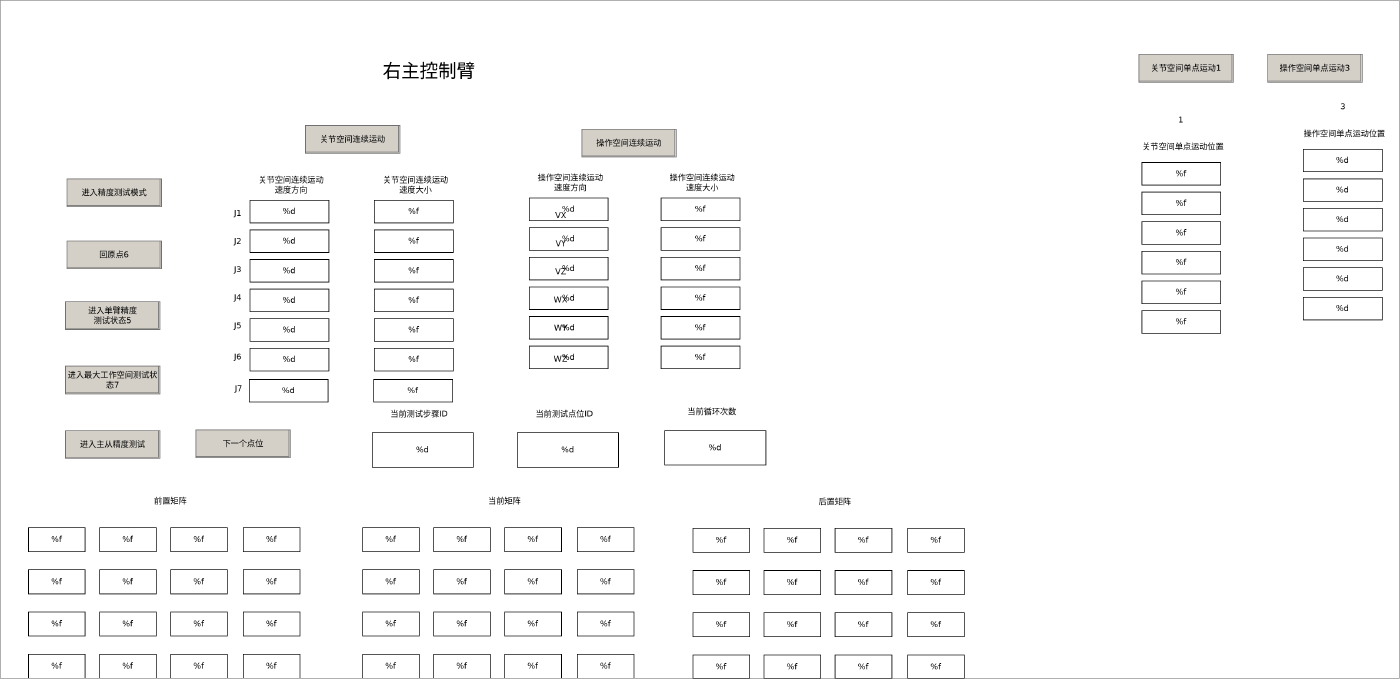
VISUALIZATION Robot_Jog_Arm2_1  // 1890x917
    Label (504,74 150x43), "右主控制臂"
    Rectangle (337,270 107x31), "%d", text variable: GVL_AccuracyTestVar.g_jntMotionDir[2][1]
        OnMouseClick: write the text variable via Default, min -1, max 1
    Label (318,235 150x29), "关节空间连续运动 速度方向"
    Rectangle (337,310 107x31), "%d", text variable: GVL_AccuracyTestVar.g_jntMotionDir[2][2]
        OnMouseClick: write the text variable via Default, min -1, max 1
    Rectangle (337,350 107x31), "%d", text variable: GVL_AccuracyTestVar.g_jntMotionDir[2][3]
        OnMouseClick: write the text variable via Default, min -1, max 1
    Rectangle (337,390 107x31), "%d", text variable: GVL_AccuracyTestVar.g_jntMotionDir[2][4]
        OnMouseClick: write the text variable via Default, min -1, max 1
    Rectangle (337,430 107x31), "%d", text variable: GVL_AccuracyTestVar.g_jntMotionDir[2][5]
        OnMouseClick: write the text variable via Default, min -1, max 1
    Rectangle (337,470 107x31), "%d", text variable: GVL_AccuracyTestVar.g_jntMotionDir[2][6]
        OnMouseClick: write the text variable via Default, min -1, max 1
    Group (1519,147 153x303), invisible if: TRUE
        Rectangle (22,72 107x31), "%f", text variable: GVL_AccuracyTestVar.g_targetJntPos[2][1]
            OnMouseClick: write the text variable via Default
        Label (3,36 150x30), "关节空间单点运动位置"
        Rectangle (22,112 107x31), "%f", text variable: GVL_AccuracyTestVar.g_targetJntPos[2][2]
            OnMouseClick: write the text variable via Default
        Rectangle (22,152 107x31), "%f", text variable: GVL_AccuracyTestVar.g_targetJntPos[2][3]
            OnMouseClick: write the text variable via Default
        Rectangle (22,192 107x31), "%f", text variable: GVL_AccuracyTestVar.g_targetJntPos[2][4]
            OnMouseClick: write the text variable via Default
        Rectangle (22,232 107x31), "%f", text variable: GVL_AccuracyTestVar.g_targetJntPos[2][5]
            OnMouseClick: write the text variable via Default
        Rectangle (22,272 107x31), "%f", text variable: GVL_AccuracyTestVar.g_targetJntPos[2][6]
            OnMouseClick: write the text variable via Default
        Label (0,0 150x30), "1"
    Rectangle (505,270 107x31), "%f", text variable: GVL_AccuracyTestVar.g_jntVel[2][1]
        OnMouseClick: write the text variable via Default
    Label (486,235 150x29), "关节空间连续运动 速度大小"
    Rectangle (505,310 107x31), "%f", text variable: GVL_AccuracyTestVar.g_jntVel[2][2]
        OnMouseClick: write the text variable via Default
    Rectangle (505,350 107x31), "%f", text variable: GVL_AccuracyTestVar.g_jntVel[2][3]
        OnMouseClick: write the text variable via Default
    Rectangle (505,390 107x31), "%f", text variable: GVL_AccuracyTestVar.g_jntVel[2][4]
        OnMouseClick: write the text variable via Default
    Rectangle (505,430 107x31), "%f", text variable: GVL_AccuracyTestVar.g_jntVel[2][5]
        OnMouseClick: write the text variable via Default
    Rectangle (505,470 107x31), "%f", text variable: GVL_AccuracyTestVar.g_jntVel[2][6]
        OnMouseClick: write the text variable via Default
    Group (1738,129 152x303), invisible if: TRUE
        Rectangle (21,72 107x31), "%d"
        Label (2,37 150x29), "操作空间单点运动位置"
        Rectangle (21,112 107x31), "%d"
        Rectangle (21,152 107x31), "%d"
        Rectangle (21,192 107x31), "%d"
        Rectangle (21,232 107x31), "%d"
        Rectangle (21,272 107x31), "%d"
        Label (0,0 150x30), "3"
    Rectangle (714,267 107x31), "%d", text variable: GVL_AccuracyTestVar.g_spatialMotionDir[2][1]
        OnMouseClick: write the text variable via Default, min -1, max 1
    Label (695,232 150x29), "操作空间连续运动 速度方向"
    Rectangle (714,307 107x31), "%d", text variable: GVL_AccuracyTestVar.g_spatialMotionDir[2][2]
        OnMouseClick: write the text variable via Default, min -1, max 1
    Rectangle (714,347 107x31), "%d", text variable: GVL_AccuracyTestVar.g_spatialMotionDir[2][3]
        OnMouseClick: write the text variable via Default, min -1, max 1
    Rectangle (714,387 107x31), "%d", text variable: GVL_AccuracyTestVar.g_spatialMotionDir[2][4]
        OnMouseClick: write the text variable via Default, min -1, max 1
    Rectangle (714,427 107x31), "%d", text variable: GVL_AccuracyTestVar.g_spatialMotionDir[2][5]
        OnMouseClick: write the text variable via Default, min -1, max 1
    Rectangle (714,467 107x31), "%d", text variable: GVL_AccuracyTestVar.g_spatialMotionDir[2][6]
        OnMouseClick: write the text variable via Default, min -1, max 1
    Rectangle (892,267 107x31), "%f", text variable: GVL_AccuracyTestVar.g_spatialVel[2][1]
        OnMouseClick: write the text variable via Default
    Label (873,232 150x29), "操作空间连续运动 速度大小"
    Rectangle (892,307 107x31), "%f", text variable: GVL_AccuracyTestVar.g_spatialVel[2][2]
        OnMouseClick: write the text variable via Default
    Rectangle (892,347 107x31), "%f", text variable: GVL_AccuracyTestVar.g_spatialVel[2][3]
        OnMouseClick: write the text variable via Default
    Rectangle (892,387 107x31), "%f", text variable: GVL_AccuracyTestVar.g_spatialVel[2][4]
        OnMouseClick: write the text variable via Default
    Rectangle (892,427 107x31), "%f", text variable: GVL_AccuracyTestVar.g_spatialVel[2][5]
        OnMouseClick: write the text variable via Default
    Rectangle (892,467 107x31), "%f", text variable: GVL_AccuracyTestVar.g_spatialVel[2][6]
        OnMouseClick: write the text variable via Default
    Button (90,241 128x38), "进入精度测试模式", colour toggle: GVL_AccuracyTestVar.g_enterPrecisionTestMode[2]
        toggle GVL_AccuracyTestVar.g_enterPrecisionTestMode[2]
    Group (1537,73 302x38), invisible if: TRUE
        Button (0,0 128x38), "关节空间单点运动1", colour toggle: A1_Arm1ModeL[2,1]
            tap A1_Arm1Mode[2,1]
        Button (174,0 128x38), "操作空间单点运动3", colour toggle: A1_Arm1ModeL[2,3]
            tap A1_Arm1Mode[2,3]
    Button (412,169 128x38), "关节空间连续运动", colour toggle: A1_Arm1ModeL[2,2]
        tap A1_Arm1Mode[2,2]
    Button (785,174 128x38), "操作空间连续运动", colour toggle: A1_Arm1ModeL[2,4]
        tap A1_Arm1Mode[2,4]
    Button (90,325 128x38), "回原点6", colour toggle: A1_Arm1ModeL[2,6]
        tap A1_Arm1Mode[2,6]
    Button (264,580 128x38), "下一个点位", colour toggle: GVL_AccuracyTestVar.g_nextStep[2]
        tap GVL_AccuracyTestVar.g_nextStep[2]
    Group (491,541 545x90)
        Rectangle (11,43 137x47), "%d", text variable: GVL_AccuracyTestVar.g_curStep[2]
        Label (0,3 150x30), "当前测试步骤ID"
        Rectangle (207,43 137x47), "%d", text variable: GVL_AccuracyTestVar.g_testPointId[2]
        Label (196,3 150x30), "当前测试点位ID"
        Rectangle (406,40 137x47), "%d", text variable: GVL_AccuracyTestVar.g_testCycleId[2]
        Label (395,0 150x30), "当前循环次数"
    Group (314,273 14x224)
        Label (0,0 14x30), "J1"
        Label (0,38 14x30), "J2"
        Label (0,76 14x30), "J3"
        Label (0,114 14x30), "J4"
        Label (0,152 14x30), "J5"
        Label (0,194 14x30), "J6"
    Group (682,276 26x224)
        Label (0,0 150x30), "VX"
        Label (0,38 150x30), "VY"
        Label (0,76 150x30), "VZ"
        Label (0,114 150x30), "WX"
        Label (0,152 150x30), "WY"
        Label (0,194 150x30), "WZ"
    Label (155,662 150x29), "前置矩阵"
    Rectangle (38,712 77x33), "%f", text variable: GVL_AccuracyTestVar.g_frontPose[2].m_rot[1,1]
    Rectangle (134,712 77x33), "%f", text variable: GVL_AccuracyTestVar.g_frontPose[2].m_rot[1,2]
    Rectangle (230,712 77x33), "%f", text variable: GVL_AccuracyTestVar.g_frontPose[2].m_rot[1,3]
    Rectangle (328,712 77x33), "%f", text variable: GVL_AccuracyTestVar.g_frontPose[2].m_pos[1]
    Rectangle (38,769 77x33), "%f", text variable: GVL_AccuracyTestVar.g_frontPose[2].m_rot[2,1]
    Rectangle (38,826 77x33), "%f", text variable: GVL_AccuracyTestVar.g_frontPose[2].m_rot[3,1]
    Rectangle (38,883 77x33), "%f", text variable: 0
    Rectangle (134,769 77x33), "%f", text variable: GVL_AccuracyTestVar.g_frontPose[2].m_rot[2,2]
    Rectangle (230,769 77x33), "%f", text variable: GVL_AccuracyTestVar.g_frontPose[2].m_rot[2,3]
    Rectangle (328,769 77x33), "%f", text variable: GVL_AccuracyTestVar.g_frontPose[2].m_pos[2]
    Rectangle (134,826 77x33), "%f", text variable: GVL_AccuracyTestVar.g_frontPose[2].m_rot[3,2]
    Rectangle (230,826 77x33), "%f", text variable: GVL_AccuracyTestVar.g_frontPose[2].m_rot[3,3]
    Rectangle (328,826 77x33), "%f", text variable: GVL_AccuracyTestVar.g_frontPose[2].m_pos[3]
    Rectangle (134,883 77x33), "%f", text variable: 0
    Rectangle (230,883 77x33), "%f", text variable: 0
    Rectangle (328,883 77x33), "%f", text variable: 1
    Label (606,662 150x29), "当前矩阵"
    Rectangle (489,712 77x33), "%f", text variable: GVL_AccuracyTestVar.g_masterArmPose[2].m_rot[1,1]
    Rectangle (585,712 77x33), "%f", text variable: GVL_AccuracyTestVar.g_masterArmPose[2].m_rot[1,2]
    Rectangle (681,712 77x33), "%f", text variable: GVL_AccuracyTestVar.g_masterArmPose[2].m_rot[1,3]
    Rectangle (779,712 77x33), "%f", text variable: GVL_AccuracyTestVar.g_masterArmPose[2].m_pos[1]
    Rectangle (489,769 77x33), "%f", text variable: GVL_AccuracyTestVar.g_masterArmPose[2].m_rot[2,1]
    Rectangle (489,826 77x33), "%f", text variable: GVL_AccuracyTestVar.g_masterArmPose[2].m_rot[3,1]
    Rectangle (489,883 77x33), "%f", text variable: 0
    Rectangle (585,769 77x33), "%f", text variable: GVL_AccuracyTestVar.g_masterArmPose[2].m_rot[2,2]
    Rectangle (681,769 77x33), "%f", text variable: GVL_AccuracyTestVar.g_masterArmPose[2].m_rot[2,3]
    Rectangle (779,769 77x33), "%f", text variable: GVL_AccuracyTestVar.g_masterArmPose[2].m_pos[2]
    Rectangle (585,826 77x33), "%f", text variable: GVL_AccuracyTestVar.g_masterArmPose[2].m_rot[3,2]
    Rectangle (681,826 77x33), "%f", text variable: GVL_AccuracyTestVar.g_masterArmPose[2].m_rot[3,3]
    Rectangle (779,826 77x33), "%f", text variable: GVL_AccuracyTestVar.g_masterArmPose[2].m_pos[3]
    Rectangle (585,883 77x33), "%f", text variable: 0
    Rectangle (681,883 77x33), "%f", text variable: 0
    Rectangle (779,883 77x33), "%f", text variable: 1
    Label (1052,663 150x29), "后置矩阵"
    Rectangle (935,713 77x33), "%f", text variable: GVL_AccuracyTestVar.g_endPose[2].m_rot[1,1]
    Rectangle (1031,713 77x33), "%f", text variable: GVL_AccuracyTestVar.g_endPose[2].m_rot[1,2]
    Rectangle (1127,713 77x33), "%f", text variable: GVL_AccuracyTestVar.g_endPose[2].m_rot[1,3]
    Rectangle (1225,713 77x33), "%f", text variable: GVL_AccuracyTestVar.g_endPose[2].m_pos[1]
    Rectangle (935,770 77x33), "%f", text variable: GVL_AccuracyTestVar.g_endPose[2].m_rot[2,1]
    Rectangle (935,827 77x33), "%f", text variable: GVL_AccuracyTestVar.g_endPose[2].m_rot[3,1]
    Rectangle (935,884 77x33), "%f", text variable: 0
    Rectangle (1031,770 77x33), "%f", text variable: GVL_AccuracyTestVar.g_endPose[2].m_rot[2,2]
    Rectangle (1127,770 77x33), "%f", text variable: GVL_AccuracyTestVar.g_endPose[2].m_rot[2,3]
    Rectangle (1225,770 77x33), "%f", text variable: GVL_AccuracyTestVar.g_endPose[2].m_pos[2]
    Rectangle (1031,827 77x33), "%f", text variable: GVL_AccuracyTestVar.g_endPose[2].m_rot[3,2]
    Rectangle (1127,827 77x33), "%f", text variable: GVL_AccuracyTestVar.g_endPose[2].m_rot[3,3]
    Rectangle (1225,827 77x33), "%f", text variable: GVL_AccuracyTestVar.g_frontPose[2].m_pos[3]
    Rectangle (1031,884 77x33), "%f", text variable: 0
    Rectangle (1127,884 77x33), "%f", text variable: 0
    Rectangle (1225,884 77x33), "%f", text variable: 1
    Button (88,407 128x38), "进入单臂精度 测试状态5", colour toggle: A1_Arm1ModeL[2,5]
        tap A1_Arm1Mode[2,5]
    Button (88,494 128x38), "进入最大工作空间测试状态7", colour toggle: A1_Arm1ModeL[2,7]
        tap A1_Arm1Mode[2,7]
    Button (88,581 128x38), "进入主从精度测试", colour toggle: GVL_AccuracyTestVar.g_MSPrecisionTest[2]
        toggle GVL_AccuracyTestVar.g_MSPrecisionTest[2]
    Label (315,510 14x30), "J7"
    Rectangle (336,512 107x31), "%d", text variable: GVL_AccuracyTestVar.g_jntMotionDir[2][7]
        OnMouseClick: write the text variable via Default, min -1, max 1
    Rectangle (504,512 107x31), "%f", text variable: GVL_AccuracyTestVar.g_jntVel[2][7]
        OnMouseClick: write the text variable via Default
END_VISUALIZATION

(* stored: Version 1.1.0.1, ProductVersion 3.1.4024.11
   Visu Robot_Jog_Arm2_1: Id {e04e2f09-56b3-4a7e-b200-a884410b2fac} *)
